{attribute 'GeneratedUsingTerminal: EL6002-0000-0016'}
{attribute addProperty BoxType "EL6002-0000-0016"}
{attribute addProperty Id "CtrlAT %Q*Ctrl_1EFB4D3B5Data_OutAT %Q*ARRAY[0..21] OF USINT22"}
{attribute addProperty CRC "3494673196"}
{attribute addProperty Size "27"}
TYPE COM_Outputs_Channel_EADA2E0D :
STRUCT
	{attribute addProperty Name "Ctrl"}
	Ctrl AT %Q* : Ctrl_1EFB4D3B;
	{attribute addProperty Name "Data_Out"}
	Data_Out AT %Q* : ARRAY[0..21] OF USINT;
END_STRUCT
END_TYPE

(* stored: Version 1.2.0.0, ProductVersion 3.1.4024.9
   DUT COM_Outputs_Channel_EADA2E0D: Id {4a79c22a-75ba-4e4a-87c0-8561efdf7d97} *)
